// TIA Portal V20 export
// export: Created 2025-12-01T14:57:06.0138851Z, ExportSetting None, DisplayName Totally Integrated Automation Portal, DisplayVersion V20 Update 3, DisplayName TIA Portal Openness, DisplayVersion V20 Update 3, DisplayName TIA Portal Version Control Interface, DisplayVersion V20 Update 3, DisplayName STEP 7 Professional, DisplayVersion V20 Update 3, DisplayName STEP 7 Safety, DisplayVersion V20 Update 2, DisplayName WinCC Basic/Comfort/Advanced, DisplayVersion V20 Update 3, DisplayName WinCC Professional, DisplayVersion V20 Update 3, DisplayName WinCC Unified, DisplayVersion V20 Update 3
FUNCTION "FC900_Reset_DB_Offset" : Void   // FC900, LAD
{ S7_Optimized_Access := 'FALSE' }
AUTHOR : GENERAL
NAME : 20130301
VERSION : 3.0
// stored: AutoNumber false, SetENOAutomatically false
   VAR_INPUT
      DB_A_RESET : DB_ANY;
      BORRAR_DESTE_BYTE : Int;
   END_VAR
   VAR_TEMP
      DESTINO : Any;
      CERO : Byte;
      BASURA : Int;
   END_VAR
BEGIN

REGION Network 1
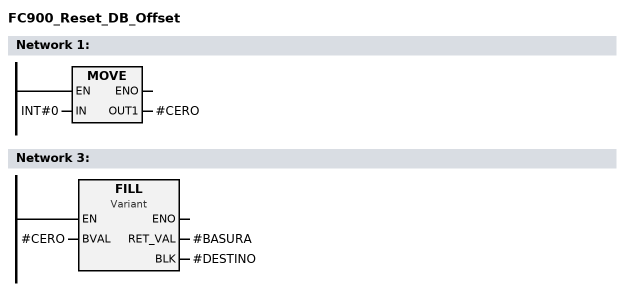
   RUNG wire#powerrail
      { S7_GenerateENO := "TRUE" } Move(in := INT#0, out1 => #CERO)
   END_RUNG
   // the same network as SCL:
   #CERO := INT#0;
END_REGION

NETWORK
TITLE = 
//ABRO EL DB PARA RESETAR Y ASI LEER SU LONGITUD
      OPN   #DB_A_RESET;
      LAR1  P##DESTINO;
// CARGAR EL ID DE SINTAXIS
      L     B#16#10;
      T     LB [AR1, P#0.0];
// CARGAR EL TIPO DE DATOS, POR DEFECTO BYTES
      L     B#16#2;
      T     LB [AR1, P#1.0];
// CARGAR LA CANTIDAD DE BYTES A COPIAR
// LEO EL TAMAÑO DEL DB A RESETAR
//COMO NO QUIERO BORRAR TODO ESTE TAMAÑO, LE RESTAMOS AL TOTAL EL OFFSET DEL QUE VAMOS A EMPEZAR
      L     DBLG;
      L     #BORRAR_DESTE_BYTE;
      -I;
      T     LW [AR1, P#2.0];
// SI ES UN DB EL ORIGEN COPIO EL NUMERO DEL DB DE DATOS
// CARGO EL NUMERO DE DB A RESETAR
      L     DBNO;
      T     LW [AR1, P#4.0];
// CARGO EL BYTE DETRABAJO
      L     #BORRAR_DESTE_BYTE;  //CON ESTO LE INDICO A PARTIR DE QUE BYTE QUIERO QUE BORRE
      SLW   3;
      T     LD [AR1, P#6.0];
// LE INDICO QUE ES UN DB
      L     B#16#84;
      T     LB [AR1, P#6.0];





REGION Network 3
   RUNG wire#powerrail
      { S7_Templates := "ptr_type := Variant" } FILL(BVAL := #CERO, RET_VAL => #BASURA, BLK => #DESTINO)
   END_RUNG
   // the same network as SCL:
   #BASURA := FILL(BVAL := #CERO, BLK => #DESTINO);
END_REGION
END_FUNCTION
